FUNCTION F_HighestReal : REAL
VAR_INPUT
	Value1																: REAL;
	Value2																: REAL;
	Value3																: REAL;
	Value4																: REAL;
END_VAR
VAR
	rValue																: REAL;
END_VAR

// F_HighestReal
// Rev 1.0 - April 25, 2024

rValue																		:= SEL(Value1 > Value2, Value2, Value1);
rValue																		:= SEL(rValue > Value3, Value3, rValue);
F_HighestReal																:= SEL(rValue > Value4, Value4, rValue);

END_FUNCTION

(* stored: Version 1.1.0.1, ProductVersion 3.1.4024.12
   POU F_HighestReal: Id {b94a2a17-5817-4fff-a828-daa4594d4b03}, SpecialFunc None *)
